FUNCTION_BLOCK FB_Encoder
VAR_OUTPUT
	fThetaMech			: LREAL;
	fOmegaMech			: LREAL;
END_VAR
VAR
	rtrig_C_status		: R_TRIG;
	fRotationDirection	: LREAL;
	fPpr				: REAL := 4096;
	fFreqScale			: REAL := 0.01;
	f16bitMax			: REAL := 65535;
	nCounter	 		: UINT;
	nCounterRaw			: UINT;
END_VAR

nCounterRaw := MAIN.stInputs.nEL5101_Counter;
nCounter := nCounterRaw * 4; // Counter is multiplied by four so we get overflow when the rotor has spinned a full circle

fThetaMech := UINT_TO_LREAL( nCounter ) / f16bitMax * 2.0 * PI; // Counter is divided by max value of UINT times two because one circle is 2pi


// Rotation direction
rtrig_C_status( CLK := MAIN.stInputs.bEl5101_C_Status );
IF rtrig_C_status.Q THEN
	IF nCounterRaw < MAIN.stInputs.nEL5101_LatchValue THEN
		fRotationDirection := -1;
	ELSIF nCounterRaw > MAIN.stInputs.nEL5101_LatchValue THEN
		fRotationDirection := 1;
	END_IF
END_IF

fOmegaMech := fRotationDirection * 2.0 * PI * ( UDINT_TO_LREAL( MAIN.stInputs.nEL5101_Frequency ) / fPpr * fFreqScale );

END_FUNCTION_BLOCK

(* stored: Version 1.1.0.1, ProductVersion 3.1.4024.11
   POU FB_Encoder: Id {6012c401-bcaa-4387-b79e-99c6207e5ca8}, SpecialFunc None *)
